(* CODESYS project Ex19.project

Project tree, tasks and I/O mapping:
  Device : CODESYS Control Win V3, 3S - Smart Software Solutions GmbH, order no. 305021, version 3.5.11.30
    application Application
      libraries: Standard, * (System)
      task MainTask (cyclic, interval t#20ms, priority 1) calls PLC_PRG
      program PLC_PRG [LD]
*)

// Device/Application/PLC_PRG
PROGRAM PLC_PRG
VAR
	I0: BYTE;
	Q0: BYTE;
	M0: BYTE;
	M1: BYTE;
END_VAR
VAR // added by the converter: edge detectors and wires of the graphical bodies
    _w1 : BOOL;
END_VAR

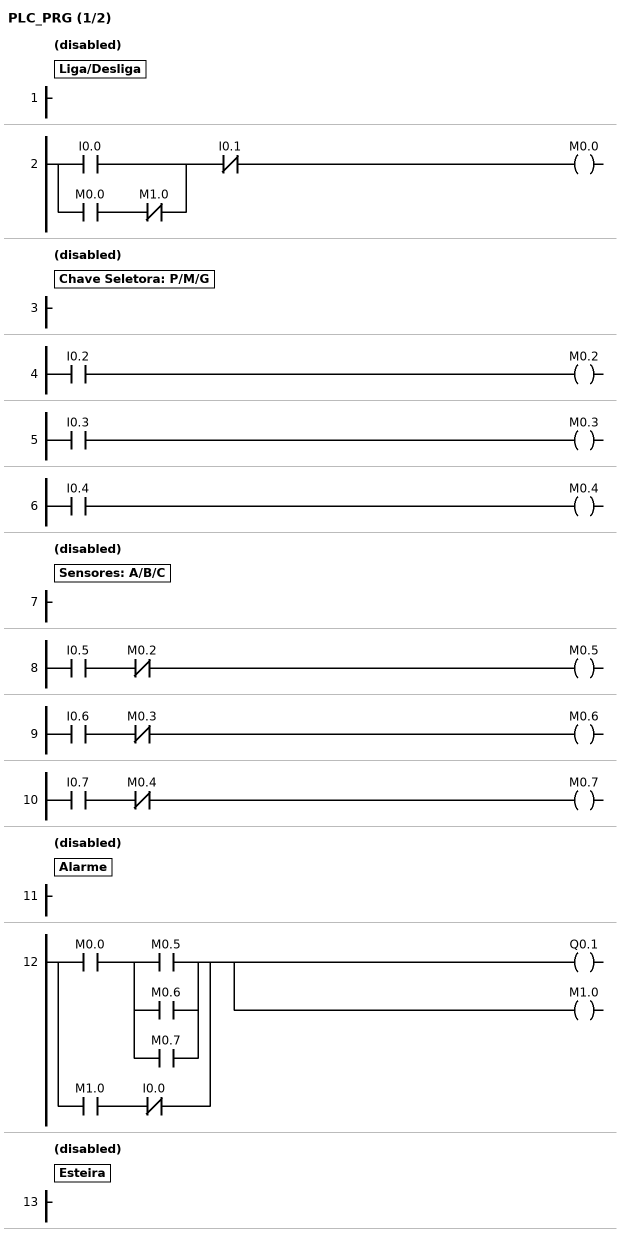
// NETWORK 1 (disabled)
// label: Liga/Desliga

// NETWORK 2
M0.0 := (I0.0 OR M0.0 AND NOT M1.0) AND NOT I0.1;

// NETWORK 3 (disabled)
// label: Chave Seletora: P/M/G

// NETWORK 4
M0.2 := I0.2;

// NETWORK 5
M0.3 := I0.3;

// NETWORK 6
M0.4 := I0.4;

// NETWORK 7 (disabled)
// label: Sensores: A/B/C

// NETWORK 8
M0.5 := I0.5 AND NOT M0.2;

// NETWORK 9
M0.6 := I0.6 AND NOT M0.3;

// NETWORK 10
M0.7 := I0.7 AND NOT M0.4;

// NETWORK 11 (disabled)
// label: Alarme

// NETWORK 12
_w1 := M0.0 AND (M0.5 OR M0.6 OR M0.7) OR M1.0 AND NOT I0.0;
Q0.1 := _w1;
M1.0 := _w1;

// NETWORK 13 (disabled)
// label: Esteira

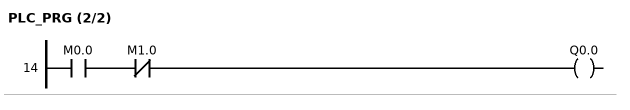
// NETWORK 14
Q0.0 := M0.0 AND NOT M1.0;

END_PROGRAM
